// TIA Portal project "indexing_station" (V16)

(* hardware
DEVICE "SCALANCE X005"  SCALANCE X-Station
   slot 0: "Switch_1"  6GK5 005-0BA00-1AB2  V1.0
   slot 0: "SCALANCE X rack"  Rail
DEVICE "ET 200SP station_1"  ET 200SP-Station
   slot 0: "IO device_1"  IM 155-6 PN/2 HF  6ES7 155-6AU01-0CN0  V4.2
   slot 0: "Rack_0"  Rack  6ES5 710-8MAx1
   slot 1: "DI 8x24VDC HF_1"  DI 8x24VDC HF  6ES7 131-6BF00-0CA0  V2.0
      slot 1: "DI 8x24VDC HF_1"  DI 8x24VDC HF
   slot 2: "DI 8x24VDC HF_2"  DI 8x24VDC HF  6ES7 131-6BF00-0CA0  V2.0
      slot 1: "DI 8x24VDC HF_2"  DI 8x24VDC HF
   slot 3: "DI 8x24VDC HF_3"  DI 8x24VDC HF  6ES7 131-6BF00-0CA0  V2.0
      slot 1: "DI 8x24VDC HF_3"  DI 8x24VDC HF
   slot 4: "DQ 8x24VDC/0.5A HF_1"  DQ 8x24VDC/0.5A HF  6ES7 132-6BF00-0CA0  V2.0
      slot 1: "DQ 8x24VDC/0.5A HF_1"  DQ 8x24VDC/0.5A HF
   slot 5: "DQ 8x24VDC/0.5A HF_2"  DQ 8x24VDC/0.5A HF  6ES7 132-6BF00-0CA0  V2.0
      slot 1: "DQ 8x24VDC/0.5A HF_2"  DQ 8x24VDC/0.5A HF
   slot 6: "Server module_1"  Server module  6ES7 193-6PA00-0AA0  V1.1
      slot 1: "Server module_1"  Server module
   slot 127: "BA 2xRJ45"  BA 2xRJ45  6ES7 193-6AR00-0AA0  V0.0
      slot 1: "Port_1"  X1 P1 R  6ES7 193-6AR00-0AA0  V0.0
      slot 2: "Port_2"  X1 P2 R  6ES7 193-6AR00-0AA0  V0.0
DEVICE "S7-1200 station_1"  S7-1200 Station
   slot 0: "Rack_0"  S7-1200 Rack  Rack  V1.0
   slot 1: "PLC_1"  CPU 1214C DC/DC/DC  6ES7 214-1AG40-0XB0  V4.4
*)

// ===== PLC "PLC_1"  CPU 1214C DC/DC/DC =====

VAR_GLOBAL   // PLC tag table "Default tag table"
   "System_Byte" AT %MB1 : Byte;
   "FirstScan" AT %M1.0 : Bool;
   "DiagStatusUpdate" AT %M1.1 : Bool;
   "AlwaysTRUE" AT %M1.2 : Bool;
   "AlwaysFALSE" AT %M1.3 : Bool;
   "Clock_Byte" AT %MB101 : Byte;
   "Clock_10Hz" AT %M101.0 : Bool;
   "Clock_5Hz" AT %M101.1 : Bool;
   "Clock_2.5Hz" AT %M101.2 : Bool;
   "Clock_2Hz" AT %M101.3 : Bool;
   "Clock_1.25Hz" AT %M101.4 : Bool;
   "Clock_1Hz" AT %M101.5 : Bool;
   "Clock_0.625Hz" AT %M101.6 : Bool;
   "Clock_0.5Hz" AT %M101.7 : Bool;
END_VAR

VAR_GLOBAL   // PLC tag table "IO_tags"
   "START BUTTON  (N.O.)" AT %I2.3 : Bool;
   "STOP BUTTON (N.C.)" AT %I2.4 : Bool;
   "EMERGENCY STOP BUTTON (N.C.)" AT %I2.5 : Bool;
   "OUTPUT POWER ON (WHITE)" AT %I2.6 : Bool;
   "INPUT 1 FROM PREVIOUS STATION" AT %I2.7 : Bool;
   "INPUT 2 FROM PREVIOUS STATION" AT %I3.0 : Bool;
   "INPUT 1 FROM NEXT STATION" AT %I3.1 : Bool;
   "INPUT 2 FROM NEXT STATION" AT %I3.2 : Bool;
   "RESET/AUTO SWITCH (RESET)" AT %I0.5 : Bool;
   "RESET/AUTO SWITCH (AUTO)" AT %I0.6 : Bool;
   "TRANSFER CYLINDER 4A RETRACTED" AT %I3.3 : Bool;
   "TRANSFER CYLINDER 4A EXTENDED" AT %I3.4 : Bool;
   "LIFT CYLINDER 1A RETRACTED" AT %I3.5 : Bool;
   "LIFT CYLINDER 1A EXTENDED" AT %I3.6 : Bool;
   "PART PRESENT (ORIENTATION POSITION)" AT %I3.7 : Bool;
   "ROTATION CYLINDER 2A RETRACTED" AT %I4.0 : Bool;
   "ROTATION CYLINDER 2A EXTENDED" AT %I4.1 : Bool;
   "SPOOL UPPER PORT DETECTED" AT %I4.2 : Bool;
   "INDEXING TABLE IN HOME POSITION" AT %I4.3 : Bool;
   "STEPPER MOTOR READY" AT %I4.4 : Bool;
   "PART PRESENT (INITIAL POSITION)" AT %I4.5 : Bool;
   "AUTOMATIC ON (GREEN)" AT %Q2.0 : Bool;
   "OUTPUT 1 TO PREVIOUS STATION" AT %Q2.1 : Bool;
   "OUTPUT 2 TO PREVIOUS STATION" AT %Q2.2 : Bool;
   "OUTPUT 1 TO NEXT STATION" AT %Q2.3 : Bool;
   "OUTPUT 2 TO NEXT STATION" AT %Q2.4 : Bool;
   "EXTEND TRANSFER CYLINDER 3A" AT %Q2.5 : Bool;
   "EXTEND LIFT CYLINDER 1A" AT %Q2.6 : Bool;
   "RETRACT LIFT CYLINDER 1A" AT %Q2.7 : Bool;
   "STEPPER MOTOR  45°" AT %Q3.0 : Bool;
   "STEPPER MOTOR 90°" AT %Q3.1 : Bool;
   "RELEASE GRIPPER 3A" AT %Q3.2 : Bool;
   "CLOSE GRIPPER 3A" AT %Q3.3 : Bool;
   "EXTEND ROTATION CYLINDER 2A" AT %Q3.4 : Bool;
   "RETRACT ROTATION CYLINDER 2A" AT %Q3.5 : Bool;
END_VAR

DATA_BLOCK "indexing_Modes Data"   // DB1
{ S7_Optimized_Access := 'TRUE' }
VERSION : 0.1
   VAR
      Automatic : Bool;
      Manual : Bool;
      Reset : Bool;
      "Pre-Automatic" : Bool;
   END_VAR
BEGIN
END_DATA_BLOCK

DATA_BLOCK "indexing_output_data"   // DB2
{ S7_Optimized_Access := 'TRUE' }
VERSION : 0.1
   VAR
      "extend transfer cylinder" : Bool;
      "extend lift cylinder_1" : Bool;
      "extend lift cylinder_2" : Bool;
      "retract lift cylinder_1" : Bool;
      "retract lift cylinder_2" : Bool;
      STEP1_MOTOR_45 : Bool;
      STEP3_MOTOR_45 : Bool;
      STEP4_MOTOR_90 : Bool;
      STEP11_MOTOR_90 : Bool;
      "release gripper" : Bool;
      "close gripper" : Bool;
      "extend rotation" : Bool;
      "retract rotation" : Bool;
      output : Bool;
   END_VAR
BEGIN
END_DATA_BLOCK

DATA_BLOCK "indexing_status Data"   // DB3
{ S7_Optimized_Access := 'TRUE' }
VERSION : 0.1
   VAR
      "CORRECT ORIENTATION" : Bool;
      STEPS : Int;
      next_step : Bool;
      previous_output : Bool;
   END_VAR
BEGIN
END_DATA_BLOCK

// folder: System blocks/Program resources

DATA_BLOCK "wait_Timer_0_DB"   // DB4
{ S7_Optimized_Access := 'TRUE' }
AUTHOR : Simatic
FAMILY : IEC
NAME : IEC_TMR
VERSION : 1.0
// stored: InstanceOfName IEC_TIMER
"IEC_TIMER"
BEGIN
END_DATA_BLOCK

DATA_BLOCK "lift_wait"   // DB5
{ S7_Optimized_Access := 'TRUE' }
AUTHOR : Simatic
FAMILY : IEC
NAME : IEC_TMR
VERSION : 1.0
// stored: InstanceOfName IEC_TIMER
"IEC_TIMER"
BEGIN
END_DATA_BLOCK

DATA_BLOCK "gripper_Timer_0_DB"   // DB6
{ S7_Optimized_Access := 'TRUE' }
AUTHOR : Simatic
FAMILY : IEC
NAME : IEC_TMR
VERSION : 1.0
// stored: InstanceOfName IEC_TIMER
"IEC_TIMER"
BEGIN
END_DATA_BLOCK

DATA_BLOCK "transfer_delay"   // DB7
{ S7_Optimized_Access := 'TRUE' }
AUTHOR : Simatic
FAMILY : IEC
NAME : IEC_TMR
VERSION : 1.0
// stored: InstanceOfName IEC_TIMER
"IEC_TIMER"
BEGIN
END_DATA_BLOCK

DATA_BLOCK "retract_delay"   // DB8
{ S7_Optimized_Access := 'TRUE' }
AUTHOR : Simatic
FAMILY : IEC
NAME : IEC_TMR
VERSION : 1.0
// stored: InstanceOfName IEC_TIMER
"IEC_TIMER"
BEGIN
END_DATA_BLOCK

DATA_BLOCK "motor90_Timer_0_DB"   // DB9
{ S7_Optimized_Access := 'TRUE' }
AUTHOR : Simatic
FAMILY : IEC
NAME : IEC_TMR
VERSION : 1.0
// stored: InstanceOfName IEC_TIMER
"IEC_TIMER"
BEGIN
END_DATA_BLOCK

DATA_BLOCK "GRIPPER_CLAMP"   // DB10
{ S7_Optimized_Access := 'TRUE' }
AUTHOR : Simatic
FAMILY : IEC
NAME : IEC_TMR
VERSION : 1.0
// stored: InstanceOfName IEC_TIMER
"IEC_TIMER"
BEGIN
END_DATA_BLOCK

// folder: (top level)

FUNCTION "indexing_modes" : Void   // FC1, LAD
TITLE = Modes Setup
{ S7_Optimized_Access := 'TRUE' }
VERSION : 0.1
BEGIN

REGION Network 1: Automatic Mode
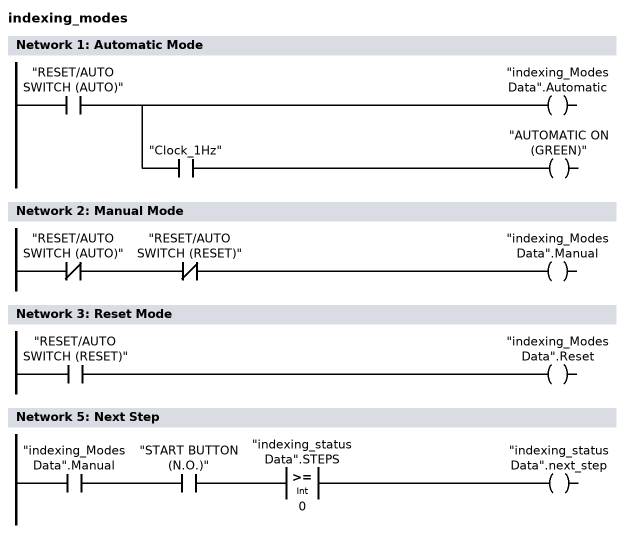
   RUNG wire#powerrail
      Contact( "RESET/AUTO SWITCH (AUTO)" )
      wire#w1
      Coil( "indexing_Modes Data".Automatic )
   END_RUNG
   RUNG wire#w1
      Contact( "Clock_1Hz" )
      Coil( "AUTOMATIC ON (GREEN)" )
   END_RUNG
   // the same network as SCL:
   "indexing_Modes Data".Automatic := "RESET/AUTO SWITCH (AUTO)";
   "AUTOMATIC ON (GREEN)" := "RESET/AUTO SWITCH (AUTO)" AND "Clock_1Hz";
END_REGION

REGION Network 2: Manual Mode
   RUNG wire#powerrail
      I_Contact( "RESET/AUTO SWITCH (AUTO)" )
      I_Contact( "RESET/AUTO SWITCH (RESET)" )
      Coil( "indexing_Modes Data".Manual )
   END_RUNG
   // the same network as SCL:
   "indexing_Modes Data".Manual := NOT "RESET/AUTO SWITCH (AUTO)" AND NOT "RESET/AUTO SWITCH (RESET)";
END_REGION

REGION Network 3: Reset Mode
   RUNG wire#powerrail
      Contact( "RESET/AUTO SWITCH (RESET)" )
      Coil( "indexing_Modes Data".Reset )
   END_RUNG
   // the same network as SCL:
   "indexing_Modes Data".Reset := "RESET/AUTO SWITCH (RESET)";
END_REGION

REGION Network 4: Pre-Automatic Mode
END_REGION

REGION Network 5: Next Step
   RUNG wire#powerrail
      Contact( "indexing_Modes Data".Manual )
      Contact( "START BUTTON  (N.O.)" )
      { S7_Templates := "SrcType := Int" } GE_Contact(in1 := "indexing_status Data".STEPS, in2 := 0)
      Coil( "indexing_status Data".next_step )
   END_RUNG
   // the same network as SCL:
   "indexing_status Data".next_step := "indexing_Modes Data".Manual AND "START BUTTON  (N.O.)" AND ("indexing_status Data".STEPS >= 0);
END_REGION
END_FUNCTION

FUNCTION "indexing_outputs" : Void   // FC2, LAD
{ S7_Optimized_Access := 'TRUE' }
VERSION : 0.1
BEGIN

REGION Network 1: Transfer Cylinder
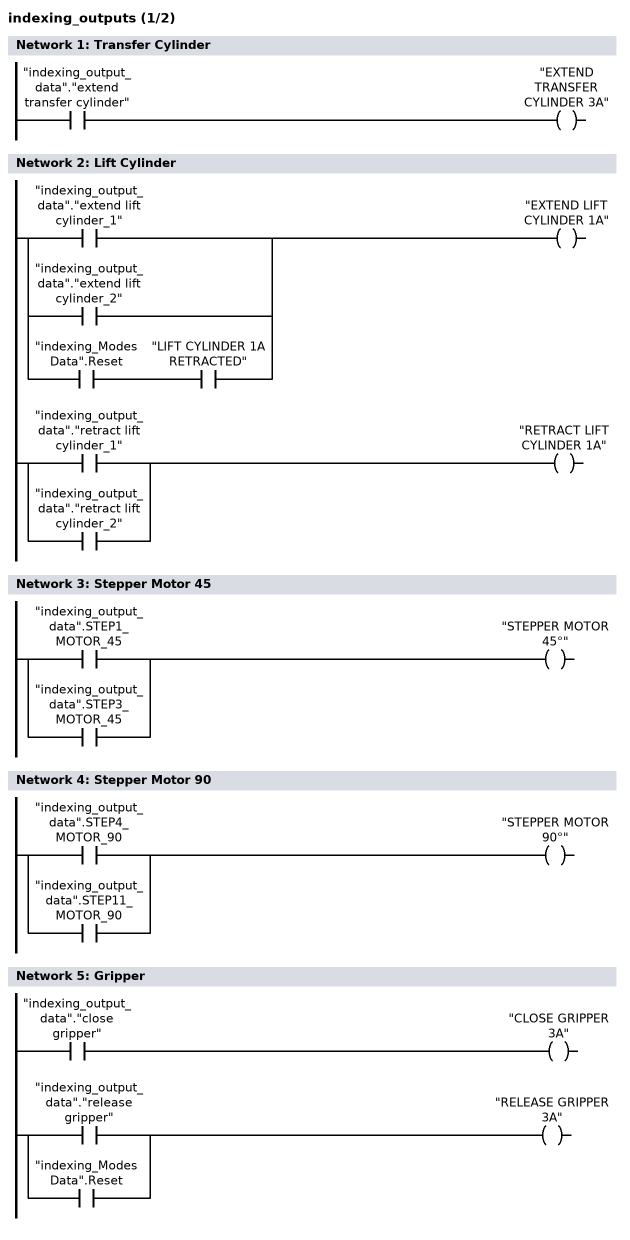
   RUNG wire#powerrail
      Contact( "indexing_output_data"."extend transfer cylinder" )
      Coil( "EXTEND TRANSFER CYLINDER 3A" )
   END_RUNG
   // the same network as SCL:
   "EXTEND TRANSFER CYLINDER 3A" := "indexing_output_data"."extend transfer cylinder";
END_REGION

REGION Network 2: Lift Cylinder
   RUNG wire#powerrail
      Contact( "indexing_output_data"."extend lift cylinder_1" )
      wire#w1
      Coil( "EXTEND LIFT CYLINDER 1A" )
   END_RUNG
   RUNG wire#powerrail
      Contact( "indexing_output_data"."extend lift cylinder_2" )
   END_RUNG wire#w1
   RUNG wire#powerrail
      Contact( "indexing_Modes Data".Reset )
      Contact( "LIFT CYLINDER 1A RETRACTED" )
   END_RUNG wire#w1
   RUNG wire#powerrail
      Contact( "indexing_output_data"."retract lift cylinder_1" )
      wire#w2
      Coil( "RETRACT LIFT CYLINDER 1A" )
   END_RUNG
   RUNG wire#powerrail
      Contact( "indexing_output_data"."retract lift cylinder_2" )
   END_RUNG wire#w2
   // the same network as SCL:
   "EXTEND LIFT CYLINDER 1A" := "indexing_output_data"."extend lift cylinder_1" OR "indexing_output_data"."extend lift cylinder_2" OR ("indexing_Modes Data".Reset AND "LIFT CYLINDER 1A RETRACTED");
   "RETRACT LIFT CYLINDER 1A" := "indexing_output_data"."retract lift cylinder_1" OR "indexing_output_data"."retract lift cylinder_2";
END_REGION

REGION Network 3: Stepper Motor 45
   RUNG wire#powerrail
      Contact( "indexing_output_data".STEP1_MOTOR_45 )
      wire#w1
      Coil( "STEPPER MOTOR  45°" )
   END_RUNG
   RUNG wire#powerrail
      Contact( "indexing_output_data".STEP3_MOTOR_45 )
   END_RUNG wire#w1
   // the same network as SCL:
   "STEPPER MOTOR  45°" := "indexing_output_data".STEP1_MOTOR_45 OR "indexing_output_data".STEP3_MOTOR_45;
END_REGION

REGION Network 4: Stepper Motor 90
   RUNG wire#powerrail
      Contact( "indexing_output_data".STEP4_MOTOR_90 )
      wire#w1
      Coil( "STEPPER MOTOR 90°" )
   END_RUNG
   RUNG wire#powerrail
      Contact( "indexing_output_data".STEP11_MOTOR_90 )
   END_RUNG wire#w1
   // the same network as SCL:
   "STEPPER MOTOR 90°" := "indexing_output_data".STEP4_MOTOR_90 OR "indexing_output_data".STEP11_MOTOR_90;
END_REGION

REGION Network 5: Gripper
   RUNG wire#powerrail
      Contact( "indexing_output_data"."close gripper" )
      Coil( "CLOSE GRIPPER 3A" )
   END_RUNG
   RUNG wire#powerrail
      Contact( "indexing_output_data"."release gripper" )
      wire#w1
      Coil( "RELEASE GRIPPER 3A" )
   END_RUNG
   RUNG wire#powerrail
      Contact( "indexing_Modes Data".Reset )
   END_RUNG wire#w1
   // the same network as SCL:
   "CLOSE GRIPPER 3A" := "indexing_output_data"."close gripper";
   "RELEASE GRIPPER 3A" := "indexing_output_data"."release gripper" OR "indexing_Modes Data".Reset;
END_REGION

REGION Network 6: Rotation Cylinder
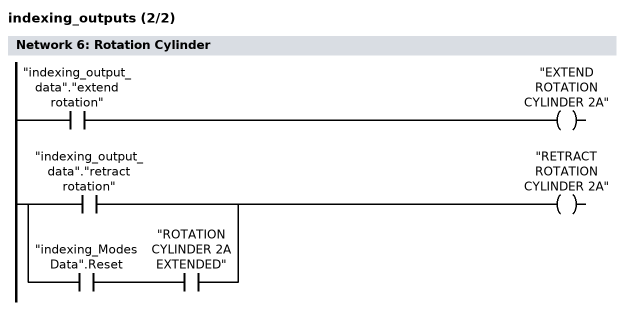
   RUNG wire#powerrail
      Contact( "indexing_output_data"."extend rotation" )
      Coil( "EXTEND ROTATION CYLINDER 2A" )
   END_RUNG
   RUNG wire#powerrail
      Contact( "indexing_output_data"."retract rotation" )
      wire#w1
      Coil( "RETRACT ROTATION CYLINDER 2A" )
   END_RUNG
   RUNG wire#powerrail
      Contact( "indexing_Modes Data".Reset )
      Contact( "ROTATION CYLINDER 2A EXTENDED" )
   END_RUNG wire#w1
   // the same network as SCL:
   "EXTEND ROTATION CYLINDER 2A" := "indexing_output_data"."extend rotation";
   "RETRACT ROTATION CYLINDER 2A" := "indexing_output_data"."retract rotation" OR ("indexing_Modes Data".Reset AND "ROTATION CYLINDER 2A EXTENDED");
END_REGION
END_FUNCTION

FUNCTION "indexing_operation" : Void   // FC3, LAD
{ S7_Optimized_Access := 'TRUE' }
VERSION : 0.1
   VAR_TEMP   // added for the SCL form of the ladder/FBD networks
      _w1 : Bool;
   END_VAR
BEGIN

REGION Network 1: STEP 1: Transfer from previous station
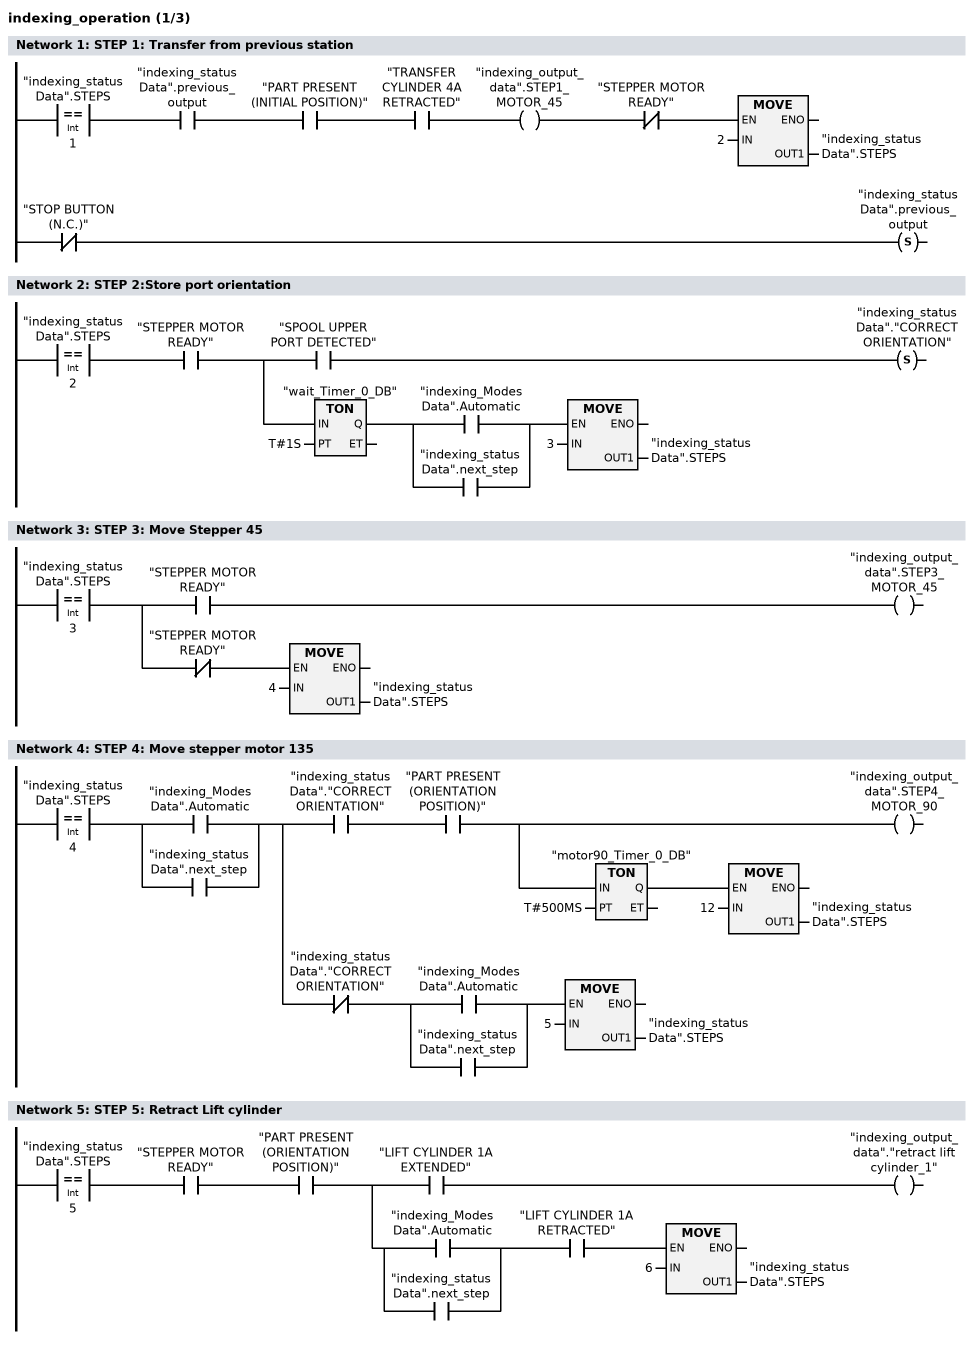
   RUNG wire#powerrail
      { S7_Templates := "SrcType := Int" } EQ_Contact(in1 := "indexing_status Data".STEPS, in2 := 1)
      Contact( "indexing_status Data".previous_output )
      Contact( "PART PRESENT (INITIAL POSITION)" )
      Contact( "TRANSFER CYLINDER 4A RETRACTED" )
      Coil( "indexing_output_data".STEP1_MOTOR_45 )
      I_Contact( "STEPPER MOTOR READY" )
      Move(in := 2, out1 => "indexing_status Data".STEPS)
   END_RUNG
   RUNG wire#powerrail
      I_Contact( "STOP BUTTON (N.C.)" )
      S_Coil( "indexing_status Data".previous_output )
   END_RUNG
   // the same network as SCL:
   "indexing_output_data".STEP1_MOTOR_45 := ("indexing_status Data".STEPS = 1) AND "indexing_status Data".previous_output AND "PART PRESENT (INITIAL POSITION)" AND "TRANSFER CYLINDER 4A RETRACTED";
   IF "indexing_output_data".STEP1_MOTOR_45 AND NOT "STEPPER MOTOR READY" THEN
       "indexing_status Data".STEPS := 2;
   END_IF;
   IF NOT "STOP BUTTON (N.C.)" THEN "indexing_status Data".previous_output := TRUE; END_IF;
END_REGION

REGION Network 2: STEP 2:Store port orientation
   #_w1 := ("indexing_status Data".STEPS = 2) AND "STEPPER MOTOR READY";
   IF #_w1 AND "SPOOL UPPER PORT DETECTED" THEN "indexing_status Data"."CORRECT ORIENTATION" := TRUE; END_IF;
   "wait_Timer_0_DB".TON(IN := #_w1, PT := T#1S);
   IF "wait_Timer_0_DB".Q AND ("indexing_Modes Data".Automatic OR "indexing_status Data".next_step) THEN
       "indexing_status Data".STEPS := 3;
   END_IF;
END_REGION

REGION Network 3: STEP 3: Move Stepper 45
   RUNG wire#powerrail
      { S7_Templates := "SrcType := Int" } EQ_Contact(in1 := "indexing_status Data".STEPS, in2 := 3)
      wire#w1
      Contact( "STEPPER MOTOR READY" )
      Coil( "indexing_output_data".STEP3_MOTOR_45 )
   END_RUNG
   RUNG wire#w1
      I_Contact( "STEPPER MOTOR READY" )
      Move(in := 4, out1 => "indexing_status Data".STEPS)
   END_RUNG
   // the same network as SCL:
   #_w1 := "indexing_status Data".STEPS = 3;
   "indexing_output_data".STEP3_MOTOR_45 := #_w1 AND "STEPPER MOTOR READY";
   IF #_w1 AND NOT "STEPPER MOTOR READY" THEN "indexing_status Data".STEPS := 4; END_IF;
END_REGION

REGION Network 4: STEP 4: Move stepper motor 135
   #_w1 := ("indexing_status Data".STEPS = 4) AND ("indexing_Modes Data".Automatic OR "indexing_status Data".next_step);
   "indexing_output_data".STEP4_MOTOR_90 := #_w1 AND "indexing_status Data"."CORRECT ORIENTATION" AND "PART PRESENT (ORIENTATION POSITION)";
   "motor90_Timer_0_DB".TON(IN := "indexing_output_data".STEP4_MOTOR_90, PT := T#500MS);
   IF "motor90_Timer_0_DB".Q THEN "indexing_status Data".STEPS := 12; END_IF;
   IF #_w1 AND NOT "indexing_status Data"."CORRECT ORIENTATION" AND ("indexing_Modes Data".Automatic OR "indexing_status Data".next_step) THEN
       "indexing_status Data".STEPS := 5;
   END_IF;
END_REGION

REGION Network 5: STEP 5: Retract Lift cylinder
   RUNG wire#powerrail
      { S7_Templates := "SrcType := Int" } EQ_Contact(in1 := "indexing_status Data".STEPS, in2 := 5)
      Contact( "STEPPER MOTOR READY" )
      Contact( "PART PRESENT (ORIENTATION POSITION)" )
      wire#w1
      Contact( "LIFT CYLINDER 1A EXTENDED" )
      Coil( "indexing_output_data"."retract lift cylinder_1" )
   END_RUNG
   RUNG wire#w1
      Contact( "indexing_Modes Data".Automatic )
      wire#w2
      Contact( "LIFT CYLINDER 1A RETRACTED" )
      Move(in := 6, out1 => "indexing_status Data".STEPS)
   END_RUNG
   RUNG wire#w1
      Contact( "indexing_status Data".next_step )
   END_RUNG wire#w2
   // the same network as SCL:
   #_w1 := ("indexing_status Data".STEPS = 5) AND "STEPPER MOTOR READY" AND "PART PRESENT (ORIENTATION POSITION)";
   "indexing_output_data"."retract lift cylinder_1" := #_w1 AND "LIFT CYLINDER 1A EXTENDED";
   IF #_w1 AND ("indexing_Modes Data".Automatic OR "indexing_status Data".next_step) AND "LIFT CYLINDER 1A RETRACTED" THEN
       "indexing_status Data".STEPS := 6;
   END_IF;
END_REGION

REGION Network 6: STEP 6: CLOSE THE GRIPPER
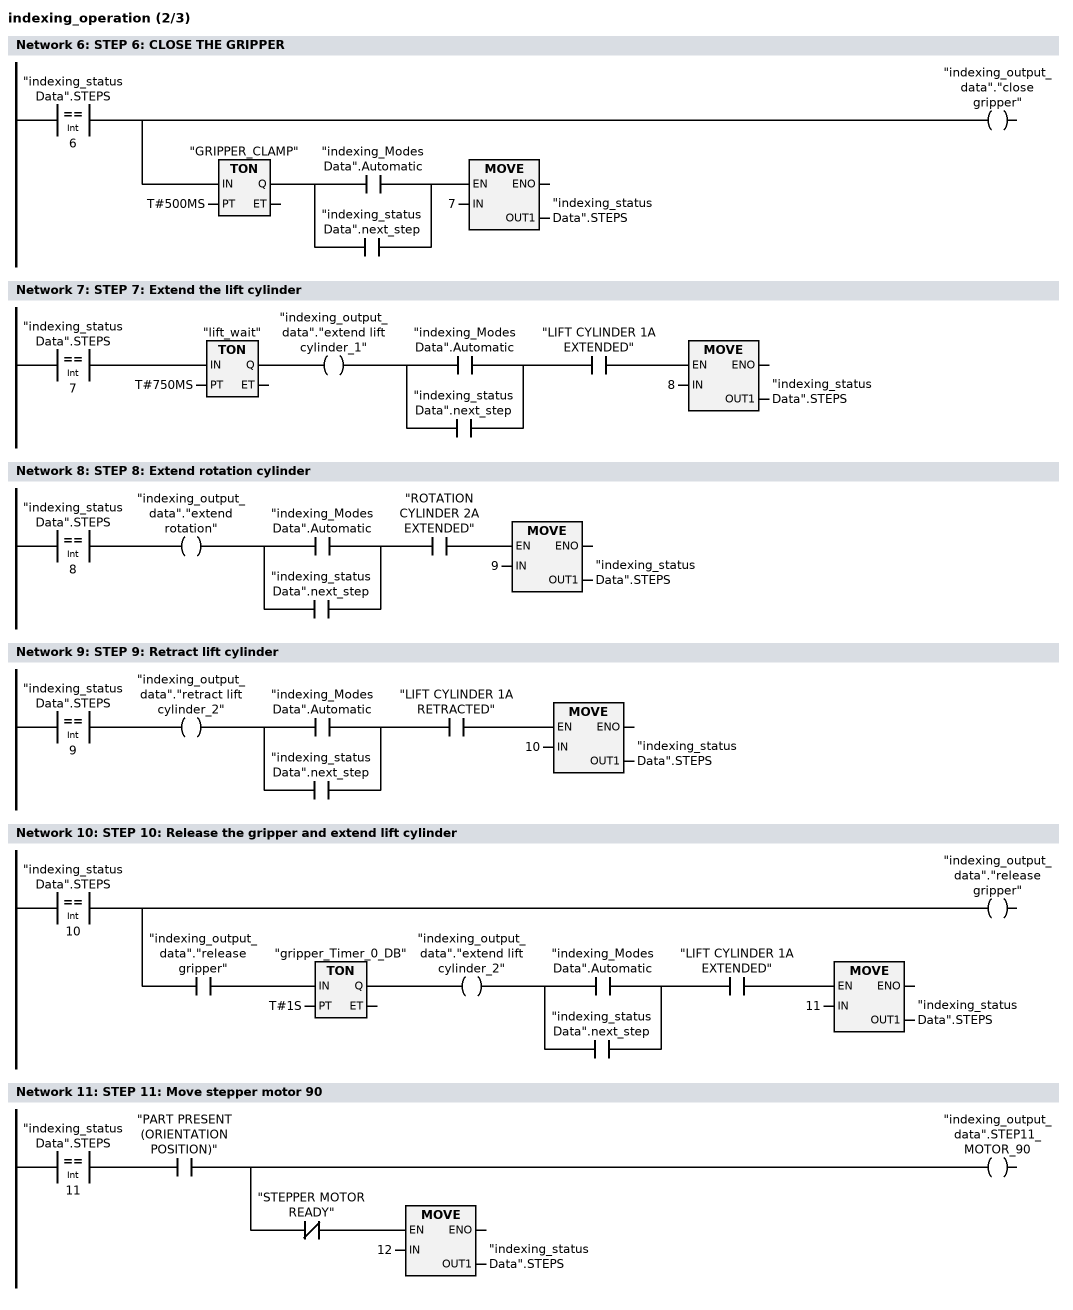
   "indexing_output_data"."close gripper" := "indexing_status Data".STEPS = 6;
   "GRIPPER_CLAMP".TON(IN := "indexing_output_data"."close gripper", PT := T#500MS);
   IF "GRIPPER_CLAMP".Q AND ("indexing_Modes Data".Automatic OR "indexing_status Data".next_step) THEN
       "indexing_status Data".STEPS := 7;
   END_IF;
END_REGION

REGION Network 7: STEP 7: Extend the lift cylinder
   "lift_wait".TON(IN := "indexing_status Data".STEPS = 7, PT := T#750MS);
   "indexing_output_data"."extend lift cylinder_1" := "lift_wait".Q;
   IF "lift_wait".Q AND ("indexing_Modes Data".Automatic OR "indexing_status Data".next_step) AND "LIFT CYLINDER 1A EXTENDED" THEN
       "indexing_status Data".STEPS := 8;
   END_IF;
END_REGION

REGION Network 8: STEP 8: Extend rotation cylinder
   RUNG wire#powerrail
      { S7_Templates := "SrcType := Int" } EQ_Contact(in1 := "indexing_status Data".STEPS, in2 := 8)
      Coil( "indexing_output_data"."extend rotation" )
      wire#w1
      Contact( "indexing_Modes Data".Automatic )
      wire#w2
      Contact( "ROTATION CYLINDER 2A EXTENDED" )
      Move(in := 9, out1 => "indexing_status Data".STEPS)
   END_RUNG
   RUNG wire#w1
      Contact( "indexing_status Data".next_step )
   END_RUNG wire#w2
   // the same network as SCL:
   "indexing_output_data"."extend rotation" := "indexing_status Data".STEPS = 8;
   IF "indexing_output_data"."extend rotation" AND ("indexing_Modes Data".Automatic OR "indexing_status Data".next_step) AND "ROTATION CYLINDER 2A EXTENDED" THEN
       "indexing_status Data".STEPS := 9;
   END_IF;
END_REGION

REGION Network 9: STEP 9: Retract lift cylinder
   RUNG wire#powerrail
      { S7_Templates := "SrcType := Int" } EQ_Contact(in1 := "indexing_status Data".STEPS, in2 := 9)
      Coil( "indexing_output_data"."retract lift cylinder_2" )
      wire#w1
      Contact( "indexing_Modes Data".Automatic )
      wire#w2
      Contact( "LIFT CYLINDER 1A RETRACTED" )
      Move(in := 10, out1 => "indexing_status Data".STEPS)
   END_RUNG
   RUNG wire#w1
      Contact( "indexing_status Data".next_step )
   END_RUNG wire#w2
   // the same network as SCL:
   "indexing_output_data"."retract lift cylinder_2" := "indexing_status Data".STEPS = 9;
   IF "indexing_output_data"."retract lift cylinder_2" AND ("indexing_Modes Data".Automatic OR "indexing_status Data".next_step) AND "LIFT CYLINDER 1A RETRACTED" THEN
       "indexing_status Data".STEPS := 10;
   END_IF;
END_REGION

REGION Network 10: STEP 10: Release the gripper and extend lift cylinder
   "indexing_output_data"."release gripper" := "indexing_status Data".STEPS = 10;
   "gripper_Timer_0_DB".TON(IN := "indexing_output_data"."release gripper" AND "indexing_output_data"."release gripper",
                           PT := T#1S);
   "indexing_output_data"."extend lift cylinder_2" := "gripper_Timer_0_DB".Q;
   IF "gripper_Timer_0_DB".Q AND ("indexing_Modes Data".Automatic OR "indexing_status Data".next_step) AND "LIFT CYLINDER 1A EXTENDED" THEN
       "indexing_status Data".STEPS := 11;
   END_IF;
END_REGION

REGION Network 11: STEP 11: Move stepper motor 90
   RUNG wire#powerrail
      { S7_Templates := "SrcType := Int" } EQ_Contact(in1 := "indexing_status Data".STEPS, in2 := 11)
      Contact( "PART PRESENT (ORIENTATION POSITION)" )
      wire#w1
      Coil( "indexing_output_data".STEP11_MOTOR_90 )
   END_RUNG
   RUNG wire#w1
      I_Contact( "STEPPER MOTOR READY" )
      Move(in := 12, out1 => "indexing_status Data".STEPS)
   END_RUNG
   // the same network as SCL:
   "indexing_output_data".STEP11_MOTOR_90 := ("indexing_status Data".STEPS = 11) AND "PART PRESENT (ORIENTATION POSITION)";
   IF "indexing_output_data".STEP11_MOTOR_90 AND NOT "STEPPER MOTOR READY" THEN
       "indexing_status Data".STEPS := 12;
   END_IF;
END_REGION

REGION Network 12: STEP 12: Extend Transfer Cylinder
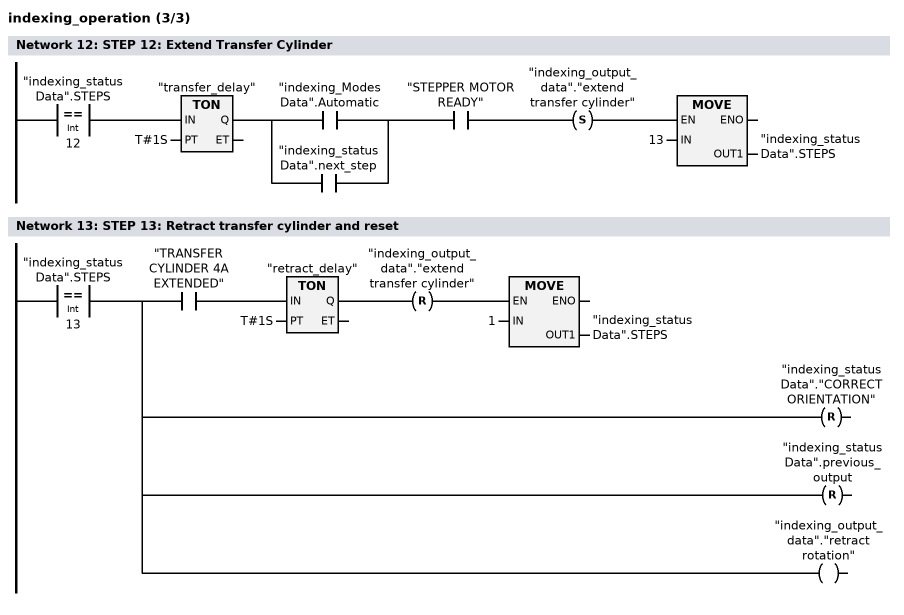
   "transfer_delay".TON(IN := "indexing_status Data".STEPS = 12, PT := T#1S);
   IF "transfer_delay".Q AND ("indexing_Modes Data".Automatic OR "indexing_status Data".next_step) AND "STEPPER MOTOR READY" THEN
       "indexing_output_data"."extend transfer cylinder" := TRUE;
       "indexing_status Data".STEPS := 13;
   END_IF;
END_REGION

REGION Network 13: STEP 13: Retract transfer cylinder and reset
   #_w1 := "indexing_status Data".STEPS = 13;
   "retract_delay".TON(IN := #_w1 AND "TRANSFER CYLINDER 4A EXTENDED", PT := T#1S);
   IF "retract_delay".Q THEN
       "indexing_output_data"."extend transfer cylinder" := FALSE;
       "indexing_status Data".STEPS := 1;
   END_IF;
   IF #_w1 THEN
       "indexing_status Data"."CORRECT ORIENTATION" := FALSE;
       "indexing_status Data".previous_output := FALSE;
   END_IF;
   "indexing_output_data"."retract rotation" := #_w1;
END_REGION
END_FUNCTION

FUNCTION "indexing_utils" : Void   // FC4, LAD
{ S7_Optimized_Access := 'TRUE' }
VERSION : 0.1
BEGIN

REGION Network 1: Modes Function
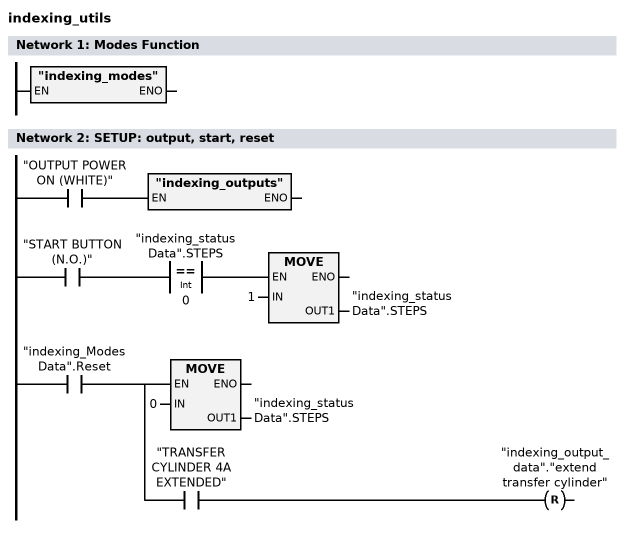
   RUNG wire#powerrail
      "indexing_modes"()
   END_RUNG
   // the same network as SCL:
   "indexing_modes"();
END_REGION

REGION Network 2: SETUP: output, start, reset
   RUNG wire#powerrail
      Contact( "OUTPUT POWER ON (WHITE)" )
      "indexing_outputs"()
   END_RUNG
   RUNG wire#powerrail
      Contact( "START BUTTON  (N.O.)" )
      { S7_Templates := "SrcType := Int" } EQ_Contact(in1 := "indexing_status Data".STEPS, in2 := 0)
      Move(in := 1, out1 => "indexing_status Data".STEPS)
   END_RUNG
   RUNG wire#powerrail
      Contact( "indexing_Modes Data".Reset )
      wire#w1
      Move(in := 0, out1 => "indexing_status Data".STEPS)
   END_RUNG
   RUNG wire#w1
      Contact( "TRANSFER CYLINDER 4A EXTENDED" )
      R_Coil( "indexing_output_data"."extend transfer cylinder" )
   END_RUNG
   // the same network as SCL:
   IF "OUTPUT POWER ON (WHITE)" THEN "indexing_outputs"(); END_IF;
   IF "START BUTTON  (N.O.)" AND ("indexing_status Data".STEPS = 0) THEN
       "indexing_status Data".STEPS := 1;
   END_IF;
   IF "indexing_Modes Data".Reset THEN "indexing_status Data".STEPS := 0; END_IF;
   IF "indexing_Modes Data".Reset AND "TRANSFER CYLINDER 4A EXTENDED" THEN
       "indexing_output_data"."extend transfer cylinder" := FALSE;
   END_IF;
END_REGION
END_FUNCTION

ORGANIZATION_BLOCK "Main"   // OB1, LAD, ProgramCycle
TITLE = "Main Program Sweep (Cycle)"
{ S7_Optimized_Access := 'TRUE' }
VERSION : 0.1
   VAR_INPUT
      Initial_Call : Bool;   // Initial call of this OB
      Remanence : Bool;   // =True, if remanent data are available
   END_VAR
BEGIN

REGION Network 1: Modes Function
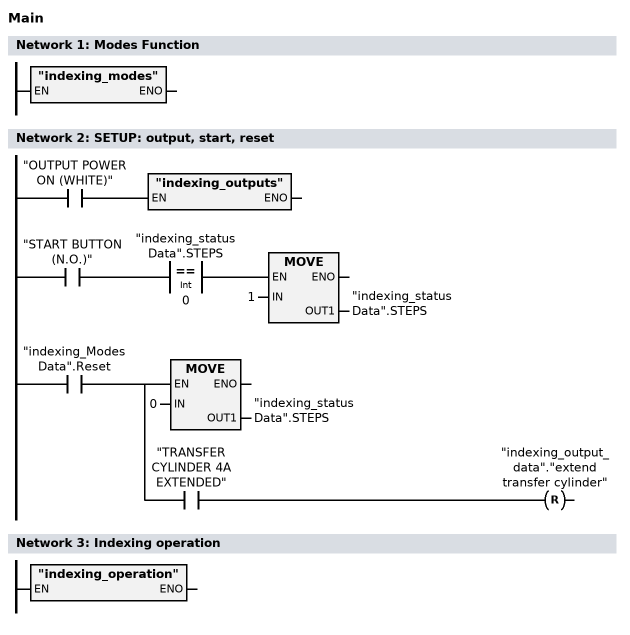
   RUNG wire#powerrail
      "indexing_modes"()
   END_RUNG
   // the same network as SCL:
   "indexing_modes"();
END_REGION

REGION Network 2: SETUP: output, start, reset
   RUNG wire#powerrail
      Contact( "OUTPUT POWER ON (WHITE)" )
      "indexing_outputs"()
   END_RUNG
   RUNG wire#powerrail
      Contact( "START BUTTON  (N.O.)" )
      { S7_Templates := "SrcType := Int" } EQ_Contact(in1 := "indexing_status Data".STEPS, in2 := 0)
      Move(in := 1, out1 => "indexing_status Data".STEPS)
   END_RUNG
   RUNG wire#powerrail
      Contact( "indexing_Modes Data".Reset )
      wire#w1
      Move(in := 0, out1 => "indexing_status Data".STEPS)
   END_RUNG
   RUNG wire#w1
      Contact( "TRANSFER CYLINDER 4A EXTENDED" )
      R_Coil( "indexing_output_data"."extend transfer cylinder" )
   END_RUNG
   // the same network as SCL:
   IF "OUTPUT POWER ON (WHITE)" THEN "indexing_outputs"(); END_IF;
   IF "START BUTTON  (N.O.)" AND ("indexing_status Data".STEPS = 0) THEN
       "indexing_status Data".STEPS := 1;
   END_IF;
   IF "indexing_Modes Data".Reset THEN "indexing_status Data".STEPS := 0; END_IF;
   IF "indexing_Modes Data".Reset AND "TRANSFER CYLINDER 4A EXTENDED" THEN
       "indexing_output_data"."extend transfer cylinder" := FALSE;
   END_IF;
END_REGION

REGION Network 3: Indexing operation
   RUNG wire#powerrail
      "indexing_operation"()
   END_RUNG
   // the same network as SCL:
   "indexing_operation"();
END_REGION
END_ORGANIZATION_BLOCK